DATA_BLOCK "Motor Control_DB"
{ S7_Optimized_Access := 'TRUE' }
VERSION : 0.1
NON_RETAIN
"Motor Control"

BEGIN

END_DATA_BLOCK

